# EPICS autosave request: iocBoot/iocDiffCtrl/auto_settings_diff_ctrl.req
file diff_ctrl.req       P=$(P), R=$(R)
